(*
SPDX-FileCopyrightText: Â© 2026 Oleksandr Tiutyk <trofimich@gmail.com>
SPDX-License-Identifier: MIT
License: https://opensource.org/license/mit
*)

(*!
<summary>Policy that ignores child critical errors.</summary>
<description>
Returns CHILD_CRITICAL_ERROR_REACTION.IGNORE, allowing the parent component to continue running without error.
</description>
*)

{attribute 'no_explicit_call' := 'do not call this function block directly'}
FUNCTION_BLOCK IgnoreChildCriticalErrorHandlingPolicy EXTENDS TOF_Core.Object IMPLEMENTS IChildCriticalErrorHandlingPolicy
VAR_STAT
	{attribute 'hide'} 
	_ClassName : STRING := __POUNAME();
END_VAR

(*!
<summary>Gets the class name of the policy.</summary>
*)
{attribute 'monitoring' := 'call'}
PROPERTY ClassName : REFERENCE TO STRING
GET
ClassName REF= _ClassName;
END_GET
END_PROPERTY

(*!
<summary>Returns CHILD_CRITICAL_ERROR_REACTION.IGNORE for the child error.</summary>
<param name="childWithError">Child component that reported the error.</param>
<param name="handlingObject">Parent component handling the failure.</param>
*)
METHOD HandleChildCriticalError : CHILD_CRITICAL_ERROR_REACTION
VAR_INPUT
	childWithError : IChildAutomationComponent;
	handlingObject : TOF_Core.IObject;
END_VAR
HandleChildCriticalError := CHILD_CRITICAL_ERROR_REACTION.IGNORE;
END_METHOD

(*!
<summary>Gets the namespace of the policy.</summary>
*)
{attribute 'monitoring' := 'call'}
PROPERTY NamespaceName : REFERENCE TO STRING
GET
NamespaceName REF= CurrentNamespace.Name;
END_GET
END_PROPERTY

(*!
<summary>Gets instance memory footprint in bytes.</summary>
*)
{attribute 'monitoring' := 'call'}
PROPERTY SelfSize : ULINT
GET
SelfSize := XSIZEOF(THIS^);
END_GET
END_PROPERTY

END_FUNCTION_BLOCK

(* stored: Version 1.1.0.1
   POU IgnoreChildCriticalErrorHandlingPolicy: Id {8369d7db-402e-4ff0-9956-4ca0be96b5af}, SpecialFunc None
   Property ClassName: Id {142d367f-52c2-4799-a090-9e9ea3fe3f2a}
   Get Get: Id {cf7261d9-980d-4bad-bb3d-b2d3720c580b}
   Method HandleChildCriticalError: Id {b99c4b31-bea4-4334-bf17-319d16a893fa}
   Property NamespaceName: Id {6689ec6c-e2d7-4dde-9c51-b7cbd56a5b4f}
   Get Get: Id {cc1242d1-31b1-49c1-b342-4678230a690e}
   Property SelfSize: Id {25bc4447-788c-47e6-99a8-6d502e8f966c}
   Get Get: Id {02ee3913-3631-492c-9cc9-adeda8a0f924} *)
